// TIA Portal V21 export
VAR_GLOBAL   // PLC tag table "Tabella delle variabili standard"
END_VAR
